(* IEC 61131-3 sources: Industry-PLC-LLM/data/PLCBEAD_repo/PLCBEAD_PLCEmbed-main/PLC-BEAD/Source/GEB/BIT_TOGGLE_W, 1 file *)

(* ---- BIT_TOGGLE_W.ST ---- *)
FUNCTION BIT_TOGGLE_W:WORD
	VAR_INPUT
		IN :	WORD;
		POS :	INT;
	END_VAR

	BIT_TOGGLE_W := SHL(WORD#1, POS) XOR IN;
END_FUNCTION

PROGRAM program0
  VAR
    LocalVar0 : WORD;
    LocalVaR1  : INT;
    CEIL5_OUT : WORD;
  END_VAR

  CEIL5_OUT := BIT_TOGGLE_W(LocalVar0, LocalVaR1 );
END_PROGRAM
